FUNCTION_BLOCK PB_NClose IMPLEMENTS I_PB
VAR
	bInput AT %I* :BOOL;
	
END_VAR

PROPERTY IsPressed : BOOL
// Property of PB button when it is pressed but for normally close
GET
IsPressed := NOT bInput;
END_GET
END_PROPERTY

PROPERTY IsReleased : BOOL
// Property of PB button when it is Released State but for normally close
GET
IsReleased := bInput;
END_GET
END_PROPERTY

END_FUNCTION_BLOCK

(* stored: Version 1.1.0.1, ProductVersion 3.1.4024.12
   POU PB_NClose: Id {a1a7af06-1a69-43db-8e36-2eb7e4bcd7bc}, SpecialFunc None
   Property IsPressed: Id {40e0ad5d-188e-46aa-9ed4-be43e8d7b340}
   Get Get: Id {4033bcc6-b0ea-4998-aa96-814f7b7ad96f}
   Property IsReleased: Id {571fd946-95ad-49f2-9584-6c4b24753cc6}
   Get Get: Id {2a8bf035-293e-448d-8ff4-3da0eb191b20} *)
